Staubli VAL3: pwrOffDrives.pgx

public program pwrOffDrives()
  local num l_i
begin
  for l_i=0 to nNUMOFAXES-1
    doEnableVoltage[l_i]=false
    doQuickStop[l_i]=false
    doSwitchOn[l_i]=false
    doEnableOp[l_i]=false
  endFor
end
